{attribute 'analysis' := '-33'}
PROGRAM INTERNAL PRG_WireFormatTests
{IF defined (UNIT_TEST)}
    fbMakeTagTests       : FB_MakeTagTests;
{END_IF}

END_PROGRAM

(* stored: Version 1.1.0.1
   POU PRG_WireFormatTests: Id {537d0474-5862-41e0-8dcf-ad6f9552d06b}, SpecialFunc None *)
